// TwinCAT 3 PLC project CraneControl
// ProgramVersion: 3.1.4023.0
// libraries:
//   Tc2_Standard, * (Beckhoff Automation GmbH)
//   Tc2_System, * (Beckhoff Automation GmbH)
//   Tc3_Module, * (Beckhoff Automation GmbH)
// project tree:
//   / GlobalTextList.TcGTLO, PlcTask.TcTTO (not stored), Visualization Manager.TcVMO (not stored)
//   MotionGeneration/FBs/ FB_AutoModeControl.TcPOU, FB_ClosedLoop.TcPOU, FB_FeedForwardAuto.TcPOU, FB_MotionGenerator.TcPOU, FB_Timer.TcPOU
//   MotionGeneration/GVL/ G_Feedbacks.TcGVL, G_MotionRef.TcGVL
//   MotionGeneration/Programs/ P_MotionGenerator.TcPOU
//   MotionGeneration/Structs/ ST_ClosedLoopParams.TcDUT, ST_MotionReferenceParams.TcDUT, ST_OpenLoopSettings.TcDUT
//   POUs/ MAIN.TcPOU
//   Simulator/HMI/ G_HMI.TcGVL, HMI_Crane.TcVIS
// real-time tasks:
//   TASK PlcTask: cycle T#10ms, priority 20, ADS port 350

// ---- MotionGeneration/Structs/ST_ClosedLoopParams.TcDUT
TYPE ST_ClosedLoopParams :
STRUCT
	fPgain : LREAL := 10.2;
	fMaxError : LREAL := 0.02; 
END_STRUCT
END_TYPE

// ---- MotionGeneration/Structs/ST_MotionReferenceParams.TcDUT
TYPE ST_MotionReferenceParams :
STRUCT
	f_x0 : LREAL;
	f_v0 : LREAL;
	f_x_ref : LREAL;
	f_v_ref : LREAL;
	f_t0 : LREAL;
	f_tRamp : LREAL;
	f_tWait : LREAL;
	f_t : LREAL; 
END_STRUCT
END_TYPE

// ---- MotionGeneration/Structs/ST_OpenLoopSettings.TcDUT
TYPE ST_OpenLoopSettings :
STRUCT
	fBoreArea : LREAL := 0.0033183;
	fAnnulusArea : LREAL := 0.0023562;
END_STRUCT
END_TYPE

// ---- MotionGeneration/GVL/G_Feedbacks.TcGVL
{attribute 'qualified_only'}
VAR_GLOBAL
	fVelFeedback : LREAL;
	fPosFeedback : LREAL; // These must come from a simulation/ROS
END_VAR

// ---- MotionGeneration/GVL/G_MotionRef.TcGVL
{attribute 'qualified_only'}
VAR_GLOBAL
	stMotionParams : ST_MotionReferenceParams := (f_x0:= 0, f_v0 := 0, f_x_ref := 0.9, f_v_ref := 0.2, f_t0 := 0.0, f_tRamp := 4.0, f_tWait := 3.0, f_t := 0.0);
	fCycleTime : LREAL := 0.01; 
	fTimer : LREAL; 
	bStart : BOOL;
	bStop : BOOL; 
	
	fMotionGeneratorPos : LREAL;
	fMotionGeneratorVel : LREAL;
	bErrorMessage : BOOL; 
	fControlledOutput : LREAL; 
	
	stOpenLoop : ST_OpenLoopSettings;
	stClosedLoop : ST_ClosedLoopParams;
	bStartOpenLoop : BOOL;
	bStartClosedLoop : BOOL; 
	
	fFeedFwdSignal : LREAL;
	fClosedLoopSignal : LREAL; 
	fClosedLoopError : LREAL; 
END_VAR

// ---- Simulator/HMI/G_HMI.TcGVL
{attribute 'qualified_only'}
VAR_GLOBAL
	bEnable : BOOL;
	bStart : BOOL;
	bStop : BOOL;
	bStartCL : BOOL;
	bStartOL : BOOL;
	bManual : BOOL;
	bAuto : BOOL; 
END_VAR

// ---- MotionGeneration/FBs/FB_AutoModeControl.TcPOU
FUNCTION_BLOCK FB_AutoModeControl
VAR_INPUT
	bEnable : BOOL;
	bStart : BOOL;
	bStop : BOOL;
	stMotionParams : ST_MotionReferenceParams;
	stClosedLoopControl : ST_ClosedLoopParams;
	stOpenLoopControl : ST_OpenLoopSettings;
	fPosFeedback : LREAL; 
END_VAR
VAR_OUTPUT
	fVelRef : LREAL;
	fPosRef : LREAL;
	fTime : LREAL;
	fPosError : LREAL;
	fCtrlOutput : LREAL;
END_VAR
VAR
	fbClock : FB_Timer;
	fbMotionRef : FB_MotionGenerator;
	fbClosedLoop : FB_ClosedLoop;
	fbOpenLoop : FB_FeedForwardAuto;
	fCtrlTemp : LREAL; 
END_VAR

IF bStart THEN
	bEnable := TRUE; 
END_IF

fbClock(bStart := G_MotionRef.bStart,
	bStop := G_MotionRef.bStop,
	fCycleTime := G_MotionRef.fCycleTime,
	fTime => G_MotionRef.fTimer); 
	
fbMotionRef(stMotionParameters := G_MotionRef.stMotionParams,
	fTimer := G_MotionRef.fTimer,
	fPosX => G_MotionRef.fMotionGeneratorPos,
	fVel => G_MotionRef.fMotionGeneratorVel,
	bError => G_MotionRef.bErrorMessage);

fbOpenLoop(bEnable := G_MotionRef.bStart,
	fVelRef := G_MotionRef.fMotionGeneratorVel,
	stOpenLoopSettings := G_MotionRef.stOpenLoop,
	fVelFeedFWD => G_MotionRef.fFeedFwdSignal); 
	
fbClosedLoop(bEnable := G_MotionRef.bStart,
	fPosRef := G_MotionRef.fMotionGeneratorPos,
	fPosFeedback := G_Feedbacks.fPosFeedback,
	stClosedLoopParams := G_MotionRef.stClosedLoop,
	stMotionParams := G_MotionRef.stMotionParams,
	fClosedLoopPosition => G_MotionRef.fClosedLoopSignal,
	fPositionError => G_MotionRef.fClosedLoopError);
	
IF bEnable THEN // This is also scaled to be between -1 and 1 to simulate a valve output
	fCtrlTemp := LIMIT(-2.0, (fbOpenLoop.fVelFeedFWD + fbClosedLoop.fClosedLoopPosition), 2.0);
	fCtrlOutput := fCtrlTemp * 60 * 3.1415/180; // full output = 60 degrees and vice verca
ELSE
	fCtrlOutput := 0;
END_IF

END_FUNCTION_BLOCK

// ---- MotionGeneration/FBs/FB_Timer.TcPOU
FUNCTION_BLOCK FB_Timer
VAR_INPUT
	bStart 		: BOOL;
	bStop 		: BOOL;
	fCycleTime  : LREAL;
END_VAR
VAR_OUTPUT
	fTime : LREAL;
END_VAR
VAR
END_VAR

IF bStart AND NOT(bStop) THEN
	fTime := fTime + fCycleTime;
ELSE
	fTime := 0.0;
END_IF

END_FUNCTION_BLOCK

// ---- MotionGeneration/FBs/FB_MotionGenerator.TcPOU
FUNCTION_BLOCK FB_MotionGenerator
VAR_INPUT
	stMotionParameters : ST_MotionReferenceParams; 
	fTimer : LREAL; 
END_VAR
VAR_OUTPUT
	fPosX : LREAL;
	fVel : LREAL;
	bError : BOOL; 
END_VAR
VAR
	f_X_SP : LREAL;
	f_vs : LREAL;
	fSlopeExt : LREAL;
	fSlopeRetr : LREAL; 
	f_as : LREAL; 
	f_sacc : LREAL; 
	f_tHold : LREAL; 
	f_t0 : LREAL;
	f_t1 : LREAL;
	f_t2 : LREAL;
	f_t3 : LREAL;
	f_t4 : LREAL;
	f_t5 : LREAL;
	f_t6 : LREAL;
	f_t7 : LREAL;
	f_x1 : LREAL;
	f_x2 : LREAL;
	f_x3 : LREAL;
	f_x4 : LREAL;
	f_x5 : LREAL; 
	f_t : LREAL; 
	
END_VAR

f_X_SP := stMotionParameters.f_x_ref - stMotionParameters.f_x0;
f_vs := stMotionParameters.f_v_ref;
f_as := f_vs/stMotionParameters.f_tRamp;
f_sacc := ((f_vs*f_vs) - (stMotionParameters.f_v0*stMotionParameters.f_v0))/f_as; 


f_tHold := (f_x_SP-f_sacc)/f_vs;

IF f_tHold < 0 THEN
	bError := TRUE;
ELSE
	bError := FALSE;
END_IF

f_t:= fTimer; 
f_t0 := stMotionParameters.f_t0;
f_t1:=stMotionParameters.f_tRamp;
f_t2:=f_tHold; 
f_t3:=stMotionParameters.f_tRamp;
f_t4:=stMotionParameters.f_tWait;
f_t5:=f_t1;
f_t6:=f_t2;
f_t7:=f_t3;

//x1 = x0 + v0*((t0+t1)-t0)-(slopeExt/t1)*((t0+t1)-t0)^2/2;
//x2 = x1 + vs*((t0+t1+t2)-(t0+t1)); 
//x4 = x_ref - v0*((t0+t1+t2+t3+t4+t5)-(t0+t1+t2+t3+t4))+(slopeRetr/t5)*((t0+t1+t2+t3+t4+t5)-(t0+t1+t2+t3+t4))^2/2; 
//x5 = x4-vs*((t0+t1+t2+t3+t4+t5+t6)-(t0+t1+t2+t3+t4+t5));  

f_x1 := stMotionParameters.f_x0 + stMotionParameters.f_v0*((f_t0 + f_t1)-f_t0) - (fSlopeExt/f_t1)*(((f_t0+f_t1)-f_t0)*((f_t0+f_t1)-f_t0))/2; 
f_x2 := f_x1 + f_vs*((f_t0+f_t1+f_t2)-(f_t0+f_t1));
f_x4 := stMotionParameters.f_x_ref - stMotionParameters.f_v0*((f_t0+f_t1+f_t2+f_t3+f_t4+f_t5)-(f_t0+f_t1+f_t2+f_t3+f_t4)) + (fSlopeRetr/f_t5)*(((f_t0+f_t1+f_t2+f_t3+f_t4+f_t5)-(f_t0+f_t1+f_t2+f_t3+f_t4))*((f_t0+f_t1+f_t2+f_t3+f_t4+f_t5)-(f_t0+f_t1+f_t2+f_t3+f_t4)))/2; 
f_x5 := f_x4 - f_vs*((f_t0+f_t1+f_t2+f_t3+f_t4+f_t5+f_t6)-(f_t0+f_t1+f_t2+f_t3+f_t4+f_t5)); 


IF bError THEN
	fPosX := stMotionParameters.f_x0;
	fVel := stMotionParameters.f_v0; 

ELSIF f_t>=0 AND f_t<f_t0 THEN
	fPosX:= stMotionParameters.f_x0; 
	fVel := stMotionParameters.f_v0;

ELSIF f_t>=f_t0 AND f_t<(f_t0+f_t1) THEN
	fPosX := stMotionParameters.f_x0 + stMotionParameters.f_v0*(f_t-f_t0)-(fSlopeExt/f_t1)*((f_t-f_t0)*(f_t-f_t0))/2;
	fVel := stMotionParameters.f_v0-(fSlopeExt/f_t1)*(f_t-f_t0);  

ELSIF f_t>=(f_t0+f_t1) AND f_t<(f_t0+f_t1+f_t2) THEN
	fPosX := f_x1 + f_vs*(f_t-(f_t0+f_t1)); 
	fVel := f_vs; 

ELSIF f_t>=(f_t0+f_t1+f_t2) AND f_t<(f_t0+f_t1+f_t2+f_t3) THEN
	fPosX := f_x2+f_vs*(f_t-(f_t0+f_t1+f_t2))+(fSlopeExt/f_t3)*((f_t-(f_t0+f_t1+f_t2))*(f_t-(f_t0+f_t1+f_t2)))/2; 
	fVel := f_vs+(fSlopeExt/f_t3)*(f_t-(f_t0+f_t1+f_t2));   

ELSIF f_t>=(f_t0+f_t1+f_t2+f_t3) AND f_t<(f_t0+f_t1+f_t2+f_t3+f_t4) THEN
	fPosX := stMotionParameters.f_x_ref;
	fVel := stMotionParameters.f_v0;  

ELSIF f_t>=(f_t0+f_t1+f_t2+f_t3+f_t4) AND f_t<(f_t0+f_t1+f_t2+f_t3+f_t4+f_t5) THEN
	fPosX := stMotionParameters.f_x_ref - stMotionParameters.f_v0*(f_t-(f_t0+f_t1+f_t2+f_t3+f_t4))+(fSlopeRetr/f_t5)*((f_t-(f_t0+f_t1+f_t2+f_t3+f_t4))*(f_t-(f_t0+f_t1+f_t2+f_t3+f_t4)))/2; 
	fVel := stMotionParameters.f_v0+(fSlopeRetr/f_t5)*(f_t-(f_t0+f_t1+f_t2+f_t3+f_t4)); 
    
ELSIF f_t>=(f_t0+f_t1+f_t2+f_t3+f_t4+f_t5) AND f_t<(f_t0+f_t1+f_t2+f_t3+f_t4+f_t5+f_t6) THEN
	fPosX := f_x4-f_vs*(f_t-(f_t0+f_t1+f_t2+f_t3+f_t4+f_t5));   
	fVel := -f_vs;    

ELSIF f_t>=(f_t0+f_t1+f_t2+f_t3+f_t4+f_t5+f_t6) AND f_t<(f_t0+f_t1+f_t2+f_t3+f_t4+f_t5+f_t6+f_t7) THEN
	fPosX := f_x5-f_vs*(f_t-(f_t0+f_t1+f_t2+f_t3+f_t4+f_t5+f_t6))-(fSlopeRetr/f_t3)*((f_t-(f_t0+f_t1+f_t2+f_t3+f_t4+f_t5+f_t6))*(f_t-(f_t0+f_t1+f_t2+f_t3+f_t4+f_t5+f_t6)))/2;    
	fVel := -f_vs-(fSlopeRetr/f_t3)*(f_t-(f_t0+f_t1+f_t2+f_t3+f_t4+f_t5+f_t6));    
 
ELSE 
	fPosX := stMotionParameters.f_x0;
	fVel := stMotionParameters.f_v0; 
END_IF

END_FUNCTION_BLOCK

// ---- MotionGeneration/FBs/FB_ClosedLoop.TcPOU
FUNCTION_BLOCK FB_ClosedLoop
VAR_INPUT
	bEnable : BOOL;
	fPosRef : LREAL;
	fPosFeedback : LREAL;
	stClosedLoopParams : ST_ClosedLoopParams; 
	stMotionParams : ST_MotionReferenceParams;
END_VAR
VAR_OUTPUT
	fClosedLoopPosition : LREAL;
	fPositionError : LREAL; 
END_VAR
VAR
	fTempPos : LREAL; 
	fTempOut : LREAL;
END_VAR

fPositionError := fPosRef - fPosFeedback; 

fTempPos := (stClosedLoopParams.fPgain * fPositionError);

IF fTempPos > 1.0 THEN // This is relevant for a valve output between 1 and -1. SHould it be used?
	fTempOut := 1;
ELSIF fTempPos >= -1.0 THEN
	fTempOut := fTempPos;
ELSE
	fTempOut := -1;
END_IF

IF bEnable THEN
	fClosedLoopPosition := fTempOut;
ELSE
	fClosedLoopPosition := 0.0; 
END_IF

END_FUNCTION_BLOCK

// ---- MotionGeneration/FBs/FB_FeedForwardAuto.TcPOU
FUNCTION_BLOCK FB_FeedForwardAuto
VAR_INPUT
	bEnable : BOOL;
	fVelRef : LREAL;
	stOpenLoopSettings : ST_OpenLoopSettings;
END_VAR
VAR_OUTPUT
	fVelFeedFWD : LREAL; 
END_VAR
VAR
	fTempOut : LREAL;
END_VAR

IF fVelRef >= 0.0 THEN
	fTempOut := stOpenLoopSettings.fBoreArea*fVelRef; // Flow to bore side
ELSE
	fTempOut := stOpenLoopSettings.fAnnulusArea * fVelRef;		// FLow to piston side
END_IF

IF bEnable THEN
	fVelFeedFWD := (60000.0*fTempOut)/150.0;
ELSE
	fVelFeedFWD := 0.0;
END_IF

END_FUNCTION_BLOCK

// ---- MotionGeneration/Programs/P_MotionGenerator.TcPOU
PROGRAM P_MotionGenerator
VAR
	fbTime : FB_Timer;
	fbGenerator : FB_MotionGenerator;
	fbAutoMode : FB_AutoModeControl;
END_VAR


G_MotionRef.bStart := G_HMI.bStart;
G_MotionRef.bStop := G_HMI.bStop;
G_MotionRef.bStartClosedLoop := G_HMI.bStartCL;
G_MotionRef.bStartOpenLoop := G_HMI.bStartOL;

//fbTime(bStart := G_MotionRef.bStart,
//	bStop := G_MotionRef.bStop,
//	fCycleTime := G_MotionRef.fCycleTime,
//	fTime => G_MotionRef.fTimer);
	
//fbGenerator(
// 	fTimer := G_MotionRef.fTimer,
//	stMotionParameters := G_MotionRef.stMotionParams,
//	fPosX => G_MotionRef.fMotionGeneratorPos,
//	fVel => G_MotionRef.fMotionGeneratorVel,
//	bError => G_MotionRef.bErrorMessage); 

fbAutoMode(bStart := G_MotionRef.bStart,
	bStop := G_MotionRef.bStop,
	stMotionParams := G_MotionRef.stMotionParams,
	stClosedLoopControl := G_MotionRef.stClosedLoop,
	stOpenLoopControl := G_MotionRef.stOpenLoop,
	fPosFeedback := G_Feedbacks.fPosFeedback,
	fCtrlOutput => G_MotionRef.fControlledOutput);

END_PROGRAM

// ---- POUs/MAIN.TcPOU
PROGRAM MAIN
VAR
	bActivateMotion : BOOL;
	fVelRef : LREAL;
	fPosRef : LREAL;
	fPosMeas : LREAL; 
	fPistonPressure : LREAL;
	fRodPressure : LREAL; 
END_VAR

P_MotionGenerator(); 
G_HMI.bStart := bActivateMotion;
fVelRef := G_MotionRef.fMotionGeneratorVel;
fPosRef := G_MotionRef.fMotionGeneratorPos;
fPosMeas := fPosRef;//G_MotionRef.fControlledOutput;
fPistonPressure := G_MotionRef.stOpenLoop.fAnnulusArea * fPosMeas;
fRodPressure := G_MotionRef.stOpenLoop.fBoreArea * fPosMeas;

END_PROGRAM

// ---- GlobalTextList.TcGTLO
TEXTLIST GlobalTextList
  24 = 'GroupBox'
END_TEXTLIST

// ---- Simulator/HMI/HMI_Crane.TcVIS
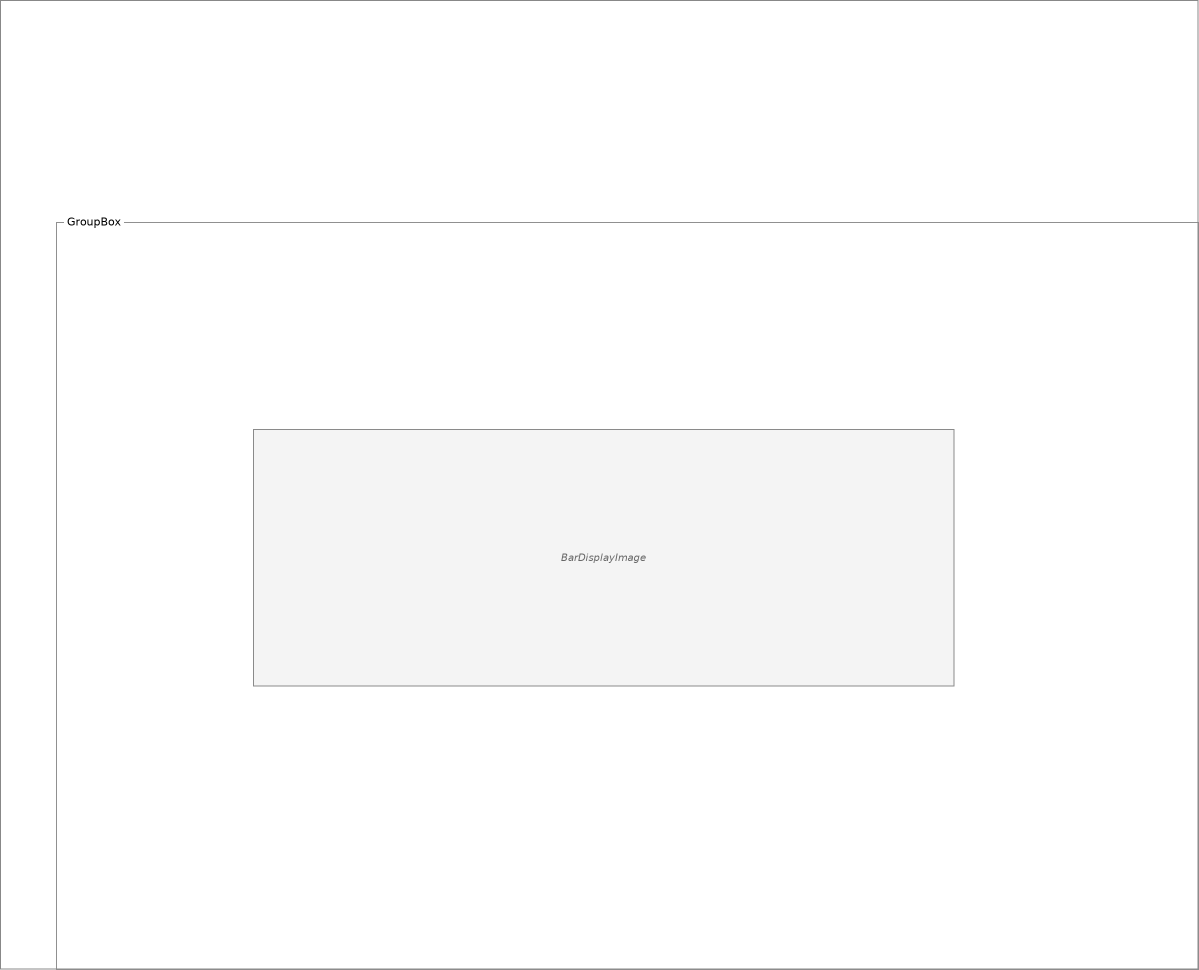
VISUALIZATION HMI_Crane  // 1199x970
    GroupBox (56,214 1143x756), "GroupBox"
        BarDisplayImage (197,215 701x257), value: G_MotionRef.fMotionGeneratorPos, style: BarDisplayImage-Gray, scale format: %.1f, scale 0..10
END_VISUALIZATION
